// TIA Portal V20 export
FUNCTION_BLOCK "FB_BwCommunication"   // FB71, SCL
{ S7_Optimized_Access := 'TRUE' }
// stored: MemoryReserve 100, SetENOAutomatically false
   VAR_INPUT
      iShuttle1Load : Bool;
      iShuttle1Unload : Bool;
      iShuttle2Load : Bool;
      iShuttle2Unload : Bool;
      iFromBwLoaderLifeFlag : Int;
      iFromBwLoaderJobDone : Bool;
      iFromBwLoaderLockShuttle : Bool;
      iFromBwLoaderDatasR : Int;
      iFromBwLoaderDatasS : Int;
      iBwInErrorState : Int;
   END_VAR
   VAR_OUTPUT
      oLifeFlagError : Bool;
      oLoadJobDone : Bool;
      oUnloadJobDone : Bool;
   END_VAR
   VAR_IN_OUT
      ioToBwLoaderLifeFlag : Int;
      ioToBwLoaderLoaderRequest { ExternalAccessible := 'False'; ExternalVisible := 'False'; ExternalWritable := 'False'} : Bool;
      ioToBwLoaderLockShuttle { ExternalAccessible := 'False'; ExternalVisible := 'False'; ExternalWritable := 'False'} : Bool;
      ioToBwLoaderDatas { ExternalAccessible := 'False'; ExternalVisible := 'False'; ExternalWritable := 'False'} : Int;
   END_VAR
   VAR
      sPrevLifeFlagFrom : Int;
      sTimerWatchdogCtrl : TON_TIME;
      sRT_1Hz { S7_SetPoint := 'True'} : R_TRIG;
      sShuttle1Locked { S7_SetPoint := 'True'} : Bool;
      sShuttle2Locked : Bool;
      sStep : Int;
      sRT_Shuttle1Load : R_TRIG;
      sRT_Shuttle1Unload : R_TRIG;
      sRT_Shuttle2Load : R_TRIG;
      sRT_Shuttle2Unload : R_TRIG;
   END_VAR
   VAR CONSTANT
      ID_SHUTTLE1_LOAD : Int := 101;
      ID_SHUTTLE1_UNLOAD : Int := 102;
      ID_SHUTTLE2_LOAD : Int := 201;
      ID_SHUTTLE2_UNLOAD : Int := 202;
   END_VAR
BEGIN
   REGION Description header 
       //==================================================================================
       // POSALUX Swiss SA / (C) Copyright 2024
       //----------------------------------------------------------------------------------
       // Title: 
       // Comment/Function: 
       //
       // Author: Fabien WALDT
       // Engineering: TIA Portal v20
       //----------------------------------------------------------------------------------
       // Change log table:
       // Version  | Date     | Expert in charge | Changes applied
       // ---------|----------|------------------|------------------------------------
       // 00.00.01 | 20260127 | WFA              | First released version
       // ==================================================================================
   END_REGION

   REGION Increment LifeFlag
       #sRT_1Hz(CLK := "Clock_1Hz");

       IF #sRT_1Hz.Q THEN
           #ioToBwLoaderLifeFlag := #ioToBwLoaderLifeFlag + 1;
       END_IF;

       IF #ioToBwLoaderLifeFlag < 0 OR #ioToBwLoaderLifeFlag > 59 THEN
           #ioToBwLoaderLifeFlag := 0;
       END_IF;
   END_REGION

   REGION Commm Control
       // Lancement du timer de controle
       #sTimerWatchdogCtrl(IN := #iFromBwLoaderLifeFlag = #sPrevLifeFlagFrom,
                           PT := T#2s);

       // Check value change
       #oLifeFlagError := FALSE;
       IF #sTimerWatchdogCtrl.Q THEN
           #oLifeFlagError := TRUE;
       END_IF;
       // Save current value
       #sPrevLifeFlagFrom := #iFromBwLoaderLifeFlag;
   END_REGION

   REGION Init
       IF  NOT #iShuttle1Load AND NOT #iShuttle1Unload AND NOT #iShuttle2Load AND NOT #iShuttle2Unload THEN
           #ioToBwLoaderDatas := 0;
               #ioToBwLoaderLoaderRequest := FALSE;
           END_IF;
   END_REGION

   REGION R_Trig Load/Unload
       #sRT_Shuttle1Load(CLK := #iShuttle1Load);
       #sRT_Shuttle1Unload(CLK := #iShuttle1Unload);
       #sRT_Shuttle2Load(CLK := #iShuttle2Load);
       #sRT_Shuttle2Unload(CLK := #iShuttle2Unload);
   END_REGION

   REGION Commm sequence

       IF NOT #oLifeFlagError THEN
           // Send Job Request
           IF #iBwInErrorState = 0 THEN
               IF #sRT_Shuttle1Load.Q THEN
                   #ioToBwLoaderDatas := #ID_SHUTTLE1_LOAD;
                   #ioToBwLoaderLoaderRequest := TRUE;
               ELSIF #sRT_Shuttle1Unload.Q THEN
                   #ioToBwLoaderDatas := #ID_SHUTTLE1_UNLOAD;
                   #ioToBwLoaderLoaderRequest := TRUE;
               ELSIF #sRT_Shuttle2Load.Q THEN
                   #ioToBwLoaderDatas := #ID_SHUTTLE2_LOAD;
                   #ioToBwLoaderLoaderRequest := TRUE;
               ELSIF #sRT_Shuttle2Unload.Q THEN
                   #ioToBwLoaderDatas := #ID_SHUTTLE2_UNLOAD;
                   #ioToBwLoaderLoaderRequest := TRUE;
               END_IF;
           END_IF;
           // Send Shuttle locked to BW
           IF #ioToBwLoaderDatas = #ID_SHUTTLE1_LOAD OR #ioToBwLoaderDatas = #ID_SHUTTLE1_UNLOAD THEN
               #ioToBwLoaderLockShuttle := "LBP_Axis05_U1".A_FDSpStop AND #iFromBwLoaderLockShuttle;
           ELSIF #ioToBwLoaderDatas = #ID_SHUTTLE2_LOAD OR #ioToBwLoaderDatas = #ID_SHUTTLE2_UNLOAD THEN
               #ioToBwLoaderLockShuttle := "LBP_Axis06_U2".A_FDSpStop AND #iFromBwLoaderLockShuttle;
               "DB_WAF".bSpy[12] := TRUE;
           ELSE
               #ioToBwLoaderLockShuttle := FALSE;
           END_IF;

           // Send Locked shuttle to axis
           IF #ioToBwLoaderLoaderRequest AND #iFromBwLoaderLockShuttle THEN
               #sShuttle1Locked := TRUE;
               #sShuttle2Locked := TRUE;
           ELSE
               #sShuttle1Locked := FALSE;
               #sShuttle2Locked := FALSE;
           END_IF;

          // Job Done
           IF #iFromBwLoaderJobDone AND (#iFromBwLoaderDatasS = #ID_SHUTTLE1_LOAD OR #iFromBwLoaderDatasS = #ID_SHUTTLE2_LOAD) THEN
               #oLoadJobDone := TRUE;
               IF "DB_LoaderShuttle1".sBwLoadUnload.sCurrent_Step_NB <> 50 AND "DB_LoaderShuttle2".sBwLoadUnload.sCurrent_Step_NB <> 50 THEN
                   #ioToBwLoaderLoaderRequest := FALSE;
               END_IF;
           ELSIF #iFromBwLoaderJobDone AND (#iFromBwLoaderDatasS = #ID_SHUTTLE1_UNLOAD OR #iFromBwLoaderDatasS = #ID_SHUTTLE2_UNLOAD) THEN
               #oUnloadJobDone := TRUE;
               IF "DB_LoaderShuttle1".sBwLoadUnload.sCurrent_Step_NB <> 150 AND "DB_LoaderShuttle2".sBwLoadUnload.sCurrent_Step_NB <> 150 THEN
                   #ioToBwLoaderLoaderRequest := FALSE;
               END_IF;
           ELSE
               #oLoadJobDone := FALSE;
               #oUnloadJobDone := FALSE;
           END_IF;
       END_IF;
   END_REGION
END_FUNCTION_BLOCK
